{attribute 'qualified_only'}
VAR_GLOBAL
END_VAR

(* stored: Version 1.1.0.1, ProductVersion 3.1.4022.7
   GVL GVL_05_Manual_Step_Motor_Other: Id {59726b0c-134a-4c65-8841-ee29288e7452} *)
